// TIA Portal V20 export
// export: Created 2025-12-01T14:57:06.6333093Z, ExportSetting None, DisplayName Totally Integrated Automation Portal, DisplayVersion V20 Update 3, DisplayName TIA Portal Openness, DisplayVersion V20 Update 3, DisplayName TIA Portal Version Control Interface, DisplayVersion V20 Update 3, DisplayName STEP 7 Professional, DisplayVersion V20 Update 3, DisplayName STEP 7 Safety, DisplayVersion V20 Update 2, DisplayName WinCC Basic/Comfort/Advanced, DisplayVersion V20 Update 3, DisplayName WinCC Professional, DisplayVersion V20 Update 3, DisplayName WinCC Unified, DisplayVersion V20 Update 3
FUNCTION "FC985_Mult_Señales_2T_Var" : Void   // FC985, LAD
{ S7_Optimized_Access := 'FALSE' }
VERSION : 3.0
// stored: AutoNumber false, SetENOAutomatically false
   VAR_INPUT
      Velocidad_0_VAR : Bool;
      Avance_T1 : Bool;
      Retroceso_T1 : Bool;
      Vel_Rapida_T1 : Bool;
      FR_Lenta_T1 : Int;
      FR_Rapida_T1 : Int;
      FR_Incremento_T1 : Int;
      Avance_T2 : Bool;
      Retroceso_T2 : Bool;
      Vel_Rapida_T2 : Bool;
      FR_Lenta_T2 : Int;
      FR_Rapida_T2 : Int;
      FR_Incremento_T2 : Int;
   END_VAR
   VAR_OUTPUT
      FR_Consigna_VAR : Int;
      FR_Incremento_VAR : Int;
   END_VAR
   VAR_IN_OUT
      Avance_Var : Bool;
      Retroceso_VAR : Bool;
      Activo_T1 : Bool;
      Activo_T2 : Bool;
   END_VAR
   VAR_TEMP   // added for the SCL form of the ladder/FBD networks
      _w1 : Bool;
   END_VAR
BEGIN

REGION Network 1
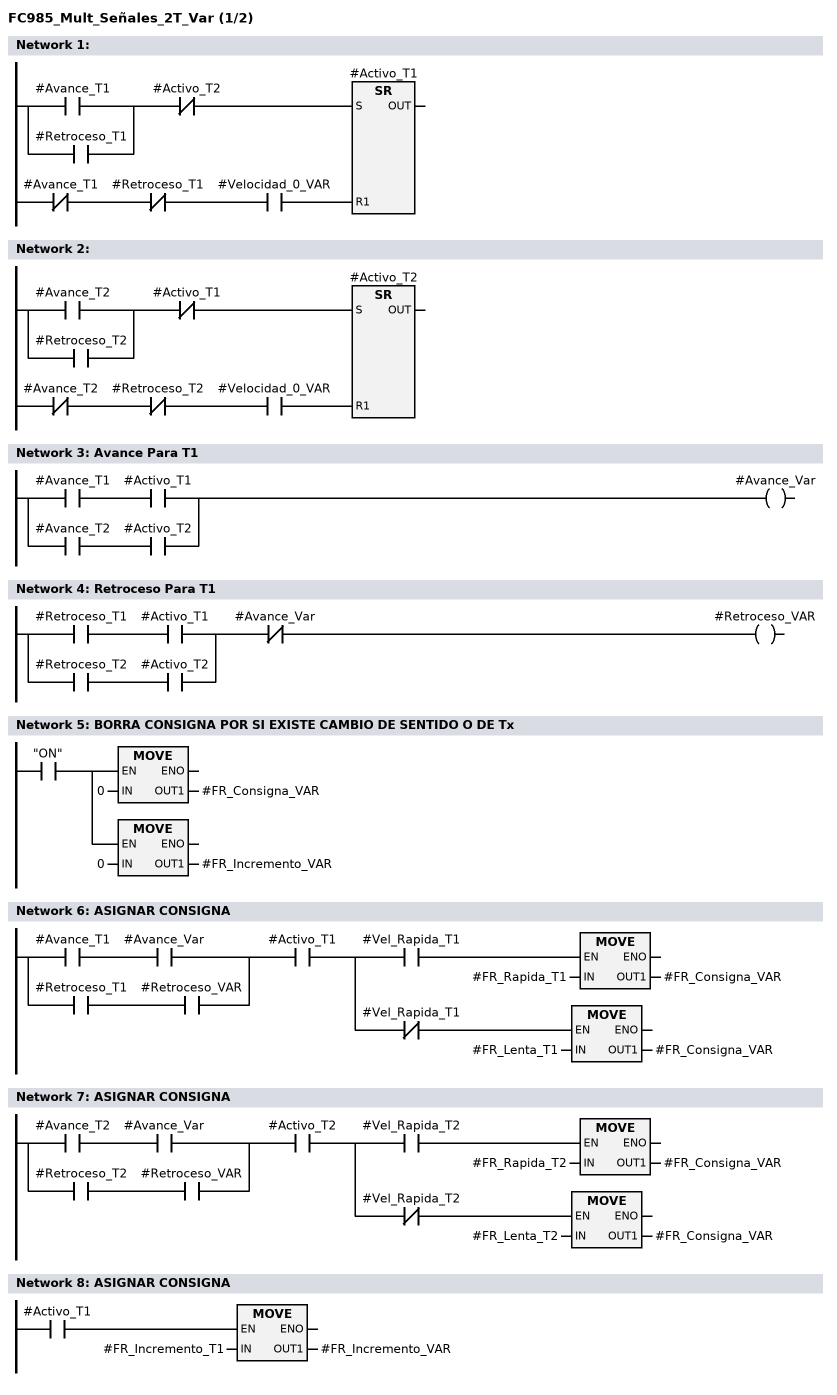
   RUNG wire#powerrail
      Contact( #Avance_T1 )
      wire#w1
      I_Contact( #Activo_T2 )
      S_SR(operand := #Activo_T1, r1 := wire#w2)
   END_RUNG
   RUNG wire#powerrail
      Contact( #Retroceso_T1 )
   END_RUNG wire#w1
   RUNG wire#powerrail
      I_Contact( #Avance_T1 )
      I_Contact( #Retroceso_T1 )
      Contact( #Velocidad_0_VAR )
   END_RUNG wire#w2
   // the same network as SCL:
   IF (#Avance_T1 OR #Retroceso_T1) AND NOT #Activo_T2 THEN
       #Activo_T1 := TRUE;   // SR flip-flop
   END_IF;
   IF NOT #Avance_T1 AND NOT #Retroceso_T1 AND #Velocidad_0_VAR THEN #Activo_T1 := FALSE; END_IF;
END_REGION

REGION Network 2
   RUNG wire#powerrail
      Contact( #Avance_T2 )
      wire#w1
      I_Contact( #Activo_T1 )
      S_SR(operand := #Activo_T2, r1 := wire#w2)
   END_RUNG
   RUNG wire#powerrail
      Contact( #Retroceso_T2 )
   END_RUNG wire#w1
   RUNG wire#powerrail
      I_Contact( #Avance_T2 )
      I_Contact( #Retroceso_T2 )
      Contact( #Velocidad_0_VAR )
   END_RUNG wire#w2
   // the same network as SCL:
   IF (#Avance_T2 OR #Retroceso_T2) AND NOT #Activo_T1 THEN
       #Activo_T2 := TRUE;   // SR flip-flop
   END_IF;
   IF NOT #Avance_T2 AND NOT #Retroceso_T2 AND #Velocidad_0_VAR THEN #Activo_T2 := FALSE; END_IF;
END_REGION

REGION Network 3: Avance Para T1
   RUNG wire#powerrail
      Contact( #Avance_T1 )
      Contact( #Activo_T1 )
      wire#w1
      Coil( #Avance_Var )
   END_RUNG
   RUNG wire#powerrail
      Contact( #Avance_T2 )
      Contact( #Activo_T2 )
   END_RUNG wire#w1
   // the same network as SCL:
   #Avance_Var := (#Avance_T1 AND #Activo_T1) OR (#Avance_T2 AND #Activo_T2);
END_REGION

REGION Network 4: Retroceso Para T1
   RUNG wire#powerrail
      Contact( #Retroceso_T1 )
      Contact( #Activo_T1 )
      wire#w1
      I_Contact( #Avance_Var )
      Coil( #Retroceso_VAR )
   END_RUNG
   RUNG wire#powerrail
      Contact( #Retroceso_T2 )
      Contact( #Activo_T2 )
   END_RUNG wire#w1
   // the same network as SCL:
   #Retroceso_VAR := ((#Retroceso_T1 AND #Activo_T1) OR (#Retroceso_T2 AND #Activo_T2)) AND NOT #Avance_Var;
END_REGION

REGION Network 5: BORRA CONSIGNA POR SI EXISTE CAMBIO DE SENTIDO O DE Tx
   RUNG wire#powerrail
      Contact( "ON" )
      wire#w1
      { S7_GenerateENO := "TRUE" } Move(in := 0, out1 => #FR_Consigna_VAR)
   END_RUNG
   RUNG wire#w1
      { S7_GenerateENO := "TRUE" } Move(in := 0, out1 => #FR_Incremento_VAR)
   END_RUNG
   // the same network as SCL:
   IF "ON" THEN
       #FR_Consigna_VAR := 0;
       #FR_Incremento_VAR := 0;
   END_IF;
END_REGION

REGION Network 6: ASIGNAR CONSIGNA
   RUNG wire#powerrail
      Contact( #Avance_T1 )
      Contact( #Avance_Var )
      wire#w1
      Contact( #Activo_T1 )
      wire#w2
      Contact( #Vel_Rapida_T1 )
      { S7_GenerateENO := "TRUE" } Move(in := #FR_Rapida_T1, out1 => #FR_Consigna_VAR)
   END_RUNG
   RUNG wire#powerrail
      Contact( #Retroceso_T1 )
      Contact( #Retroceso_VAR )
   END_RUNG wire#w1
   RUNG wire#w2
      I_Contact( #Vel_Rapida_T1 )
      { S7_GenerateENO := "TRUE" } Move(in := #FR_Lenta_T1, out1 => #FR_Consigna_VAR)
   END_RUNG
   // the same network as SCL:
   #_w1 := ((#Avance_T1 AND #Avance_Var) OR (#Retroceso_T1 AND #Retroceso_VAR)) AND #Activo_T1;
   IF #_w1 AND #Vel_Rapida_T1 THEN #FR_Consigna_VAR := #FR_Rapida_T1; END_IF;
   IF #_w1 AND NOT #Vel_Rapida_T1 THEN #FR_Consigna_VAR := #FR_Lenta_T1; END_IF;
END_REGION

REGION Network 7: ASIGNAR CONSIGNA
   RUNG wire#powerrail
      Contact( #Avance_T2 )
      Contact( #Avance_Var )
      wire#w1
      Contact( #Activo_T2 )
      wire#w2
      Contact( #Vel_Rapida_T2 )
      { S7_GenerateENO := "TRUE" } Move(in := #FR_Rapida_T2, out1 => #FR_Consigna_VAR)
   END_RUNG
   RUNG wire#powerrail
      Contact( #Retroceso_T2 )
      Contact( #Retroceso_VAR )
   END_RUNG wire#w1
   RUNG wire#w2
      I_Contact( #Vel_Rapida_T2 )
      { S7_GenerateENO := "TRUE" } Move(in := #FR_Lenta_T2, out1 => #FR_Consigna_VAR)
   END_RUNG
   // the same network as SCL:
   #_w1 := ((#Avance_T2 AND #Avance_Var) OR (#Retroceso_T2 AND #Retroceso_VAR)) AND #Activo_T2;
   IF #_w1 AND #Vel_Rapida_T2 THEN #FR_Consigna_VAR := #FR_Rapida_T2; END_IF;
   IF #_w1 AND NOT #Vel_Rapida_T2 THEN #FR_Consigna_VAR := #FR_Lenta_T2; END_IF;
END_REGION

REGION Network 8: ASIGNAR CONSIGNA
   RUNG wire#powerrail
      Contact( #Activo_T1 )
      { S7_GenerateENO := "TRUE" } Move(in := #FR_Incremento_T1, out1 => #FR_Incremento_VAR)
   END_RUNG
   // the same network as SCL:
   IF #Activo_T1 THEN #FR_Incremento_VAR := #FR_Incremento_T1; END_IF;
END_REGION

REGION Network 9: ASIGNAR CONSIGNA
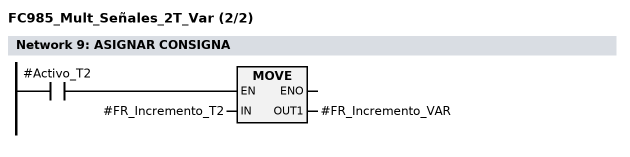
   RUNG wire#powerrail
      Contact( #Activo_T2 )
      { S7_GenerateENO := "TRUE" } Move(in := #FR_Incremento_T2, out1 => #FR_Incremento_VAR)
   END_RUNG
   // the same network as SCL:
   IF #Activo_T2 THEN #FR_Incremento_VAR := #FR_Incremento_T2; END_IF;
END_REGION
END_FUNCTION
